/// configuration data that is used during boot to configure the Units equipment
TYPE MachineDataConfig :
STRUCT
  Simulated : BOOL;
END_STRUCT
END_TYPE

(* stored: Version 1.1.0.1
   DUT MachineDataConfig: Id {f3031aed-ae83-4d0a-a5fe-f0794217a184} *)
